// TIA Portal V17 export
// export: Created 2021-12-03T08:08:09.0167679Z, ExportSetting WithDefaults, DisplayName Totally Integrated Automation Portal, DisplayVersion V17, DisplayName TIA Portal Openness, DisplayVersion V17, DisplayName TIA Portal Version Control Interface, DisplayVersion V17, DisplayName STEP 7 Professional, DisplayVersion V17, DisplayName STEP 7 Safety, DisplayVersion V17, DisplayName WinCC Advanced, DisplayVersion V17
VAR_GLOBAL   // PLC tag table "HMI_Log"
   SafetyPer AT %MW300 : Word;
   SafetyPer_0 AT %M300.0 : Bool;
   SafetyPer_1 AT %M300.1 : Bool;
   SafetyPer_2 AT %M300.2 : Bool;
   SafetyPer_3 AT %M300.3 : Bool;
   SafetyPer_4 AT %M300.4 : Bool;
   SafetyPer_5 AT %M300.5 : Bool;
   SafetyPer_6 AT %M300.6 : Bool;
   SafetyPer_7 AT %M300.7 : Bool;
   SafetyPer_8 AT %M301.0 : Bool;
   SafetyPer_9 AT %M301.1 : Bool;
   SafetyPer_10 AT %M301.2 : Bool;
   SafetyPer_11 AT %M301.3 : Bool;
   SafetyPer_12 AT %M301.4 : Bool;
   SafetyPer_13 AT %M301.5 : Bool;
   SafetyPer_14 AT %M301.6 : Bool;
   SafetyPer_15 AT %M301.7 : Bool;
   ScanSeqCond AT %MW302 : Word;
   ScanSeqCond_0 AT %M302.0 : Bool;
   ScanSeqCond_1 AT %M302.1 : Bool;
   ScanSeqCond_2 AT %M302.2 : Bool;
   ScanSeqCond_3 AT %M302.3 : Bool;
   ScanSeqCond_4 AT %M302.4 : Bool;
   ScanSeqCond_5 AT %M302.5 : Bool;
   ScanSeqCond_6 AT %M302.6 : Bool;
   ScanSeqCond_7 AT %M302.7 : Bool;
   ScanSeqCond_8 AT %M303.0 : Bool;
   ScanSeqCond_9 AT %M303.1 : Bool;
   ScanSeqCond_10 AT %M303.2 : Bool;
   ScanSeqCond_11 AT %M303.3 : Bool;
   ScanSeqCond_12 AT %M303.4 : Bool;
   ScanSeqCond_13 AT %M303.5 : Bool;
   ScanSeqCond_14 AT %M303.6 : Bool;
   ScanSeqCond_15 AT %M303.7 : Bool;
END_VAR
